FUNCTION_BLOCK CRANE2_FOLLOW_MACHINE (* Service Interface Function Block Type *)
  (* Standard: 61499-2 *)
  (* Version 1.0, 2019-01-24, iotdeveloperpk *)
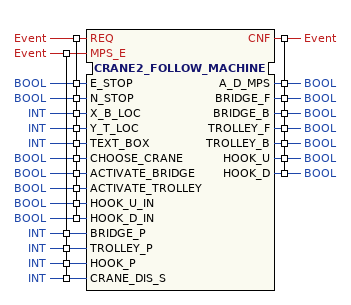
  EVENT_INPUT
    REQ WITH E_STOP, N_STOP, X_B_LOC, Y_T_LOC, TEXT_BOX, ACTIVATE_BRIDGE, ACTIVATE_TROLLEY, HOOK_U_IN, CHOOSE_CRANE, HOOK_D_IN; (* Service Request *)
    MPS_E WITH BRIDGE_P, TROLLEY_P, HOOK_P, CRANE_DIS_S;
  END_EVENT
  EVENT_OUTPUT
    CNF WITH A_D_MPS, BRIDGE_F, BRIDGE_B, TROLLEY_F, TROLLEY_B, HOOK_U, HOOK_D; (* Confirmation of Requested Service *)
  END_EVENT
  VAR_INPUT
    E_STOP : BOOL;
    N_STOP : BOOL;
    X_B_LOC : INT;
    Y_T_LOC : INT;
    TEXT_BOX : INT;
    CHOOSE_CRANE : BOOL;
    ACTIVATE_BRIDGE : BOOL;
    ACTIVATE_TROLLEY : BOOL;
    HOOK_U_IN : BOOL;
    HOOK_D_IN : BOOL;
    BRIDGE_P : INT;
    TROLLEY_P : INT;
    HOOK_P : INT;
    CRANE_DIS_S : INT;
  END_VAR
  VAR_OUTPUT
    A_D_MPS : BOOL;
    BRIDGE_F : BOOL;
    BRIDGE_B : BOOL;
    TROLLEY_F : BOOL;
    TROLLEY_B : BOOL;
    HOOK_U : BOOL;
    HOOK_D : BOOL;
  END_VAR
  SERVICE APPLICATION/RESOURCE (* Service Interface Function Block Type *)
    SEQUENCE normal_establishment
      APPLICATION.INIT+(PARAMS) -> RESOURCE.initialize(PARAMS) -> APPLICATION.INITO+();
    END_SEQUENCE
    SEQUENCE unsuccessful_establishment
      APPLICATION.INIT+(PARAMS) -> RESOURCE.initialize(PARAMS) -> APPLICATION.INITO-(STATUS);
    END_SEQUENCE
    SEQUENCE request_confirm
      APPLICATION.REQ+(SD) -> RESOURCE.request(SD) -> APPLICATION.CNF+(RD);
    END_SEQUENCE
    SEQUENCE request_inhibited
      APPLICATION.REQ-(SD) -> APPLICATION.CNF-(STATUS);
    END_SEQUENCE
    SEQUENCE request_error
      APPLICATION.REQ+(SD) -> RESOURCE.request(SD) -> APPLICATION.CNF-(STATUS);
    END_SEQUENCE
    SEQUENCE indication_response
      RESOURCE.indicate(RD) -> APPLICATION.IND+(RD);
      APPLICATION.RSP(QI,SD) -> RESOURCE.response(QI,SD);
    END_SEQUENCE
    SEQUENCE indication_inhibited
      RESOURCE.indicate(RD,QI=FALSE) -> RESOURCE.inhibited();
    END_SEQUENCE
    SEQUENCE error_indication
      RESOURCE.error(STATUS) -> APPLICATION.IND-(STATUS);
    END_SEQUENCE
    SEQUENCE application_initiated_termination
      APPLICATION.INIT-() -> RESOURCE.terminate() -> APPLICATION.INITO-(STATUS);
    END_SEQUENCE
    SEQUENCE resource_initiated_termination
      -> APPLICATION.INITO-(STATUS);
    END_SEQUENCE
  END_SERVICE
END_FUNCTION_BLOCK
